FUNCTION_BLOCK AdjustableSizeReplyRpcHandler IMPLEMENTS I_RpcHandler
VAR
END_VAR

METHOD Handle
VAR_INPUT
	Parameters : I_RpcParameters;
	Response : I_SynchronousRpcResponse;
END_VAR
VAR
	size : UDINT;
	pBytes : POINTER TO BYTE;
END_VAR
IF NOT Parameters.TryGetParameter('Size',size) THEN
	Response.RejectWithMessage('Missing Size parameter');
	RETURN;
END_IF

IF size = 0 THEN 
	Response.CompleteWithNull();
END_IF

pBytes := __NEW(BYTE, size);
memset(pBytes, 1, size);

Response.CompleteWithBytesAsHex(pBytes, size);

__Delete(pBytes);
END_METHOD

END_FUNCTION_BLOCK

(* stored: Version 1.1.0.1, ProductVersion 3.1.4024.12
   POU AdjustableSizeReplyRpcHandler: Id {9299e15a-1853-4d5c-887c-44fb5a606abe}, SpecialFunc None
   Method Handle: Id {9f2bbb3b-e3e7-4379-9b54-5579b5c73f06} *)
